{attribute 'qualified_only'}
VAR_GLOBAL
	P1 AT %Q*: BOOL;	// Meldeleuchte Störung
	P2 AT %Q*: BOOL;	// Meldeleuchte Betrieb
	P3 AT %Q*: BOOL;	// Meldeleuchte Füllstand Min.
	Q1 AT %Q*: BOOL;	// Motorschütz Pumpe 1
	Q2 AT %Q*: BOOL;	// Motorschütz Pumpe 2
END_VAR

(* stored: Version 1.1.0.1, ProductVersion 3.1.4024.4
   GVL SimDA: Id {efa3d63a-96e1-4204-b1e7-9f3703bd4f03} *)
